// TIA Portal V20 export
TYPE "typeSequenceControlNodeHomeCheck_jrOutPnPLeft"
// stored: Namespace Unit1.Em2
   STRUCT
      partNoDetect { ExternalWritable := 'False'} : Bool;
      partDetect { ExternalWritable := 'False'} : Bool;
   END_STRUCT;
END_TYPE
